Omron CX-Programmer project NewProject (CX-Programmer 9.61)

# PLC NewPLC1: CJ2M CPU11
I/O table (CPU CJ2M-CPU11): rack 0 slot 0 CJ1W-ID211; rack 0 slot 1 CJ1W-OD211

## Global symbols (name address type ; comment)
0.00 BOOL  ; PB Start
0.01 BOOL  ; PB Stop
0.02 BOOL  ; Emergency Stop
0.04 BOOL  ; Sensor C2PE
0.05 BOOL  ; PB1 C1
0.06 BOOL  ; PB2 C1
0.07 BOOL  ; Sensor STPX1
0.08 BOOL  ; Sensor STPX2
0.09 BOOL  ; Sensor STPX3
0.10 BOOL  ; Sensor PECA
0.11 BOOL  ; Sensor PECB
0.12 BOOL  ; Sensor PECC
0.14 BOOL  ; Sensor PEST
0.15 BOOL  ; Reset
1.00 BOOL  ; Conveyor C1
1.01 BOOL  ; Conveyor C2
1.02 BOOL  ; Light PBC1
1.03 BOOL  ; LIght PBC2
1.04 BOOL  ; Buzzer
1.06 BOOL  ; Conveyor ST2
1.07 BOOL  ; Coveyor CA
1.08 BOOL  ; Coveyor CB
1.09 BOOL  ; Conveyor CC
1.10 BOOL  ; Indikator Lampu CA
1.11 BOOL  ; Indikator Lampu CB
1.13 BOOL  ; Indikator Lampu CC
2.00 BOOL  ; System ON
2.01 BOOL  ; Memory 2
2.02 BOOL  ; Memory 3
2.03 BOOL  ; Masuk ke CA
2.04 BOOL  ; Masuk ke CB
2.05 BOOL  ; Masuk ke CC
D1 CHANNEL  ; Barcode Scanner
D100 CHANNEL  ; Data Barcode
D101 CHANNEL  ; Posisi Mobil
D102 CHANNEL  ; Conveyor ST2
T0000 BOOL  ; TB PBC2 UP
T0001 BOOL  ; TB PBC1 UP
T0002 BOOL  ; TB PBC2 DOWN
T0003 BOOL  ; TB PBC1 DOWN
T0004 BOOL  ; T BUZZ PB1/2 C1
T0005 BOOL  ; T BUZZ C15s
BarcodeProcess BarcodeScanner
Menentukan_Posisi_STPX SensorSTPX
Pengiriman PengirimanKeCACBCC

## Program SesiC (cyclic task 0)

### Section Main_Program

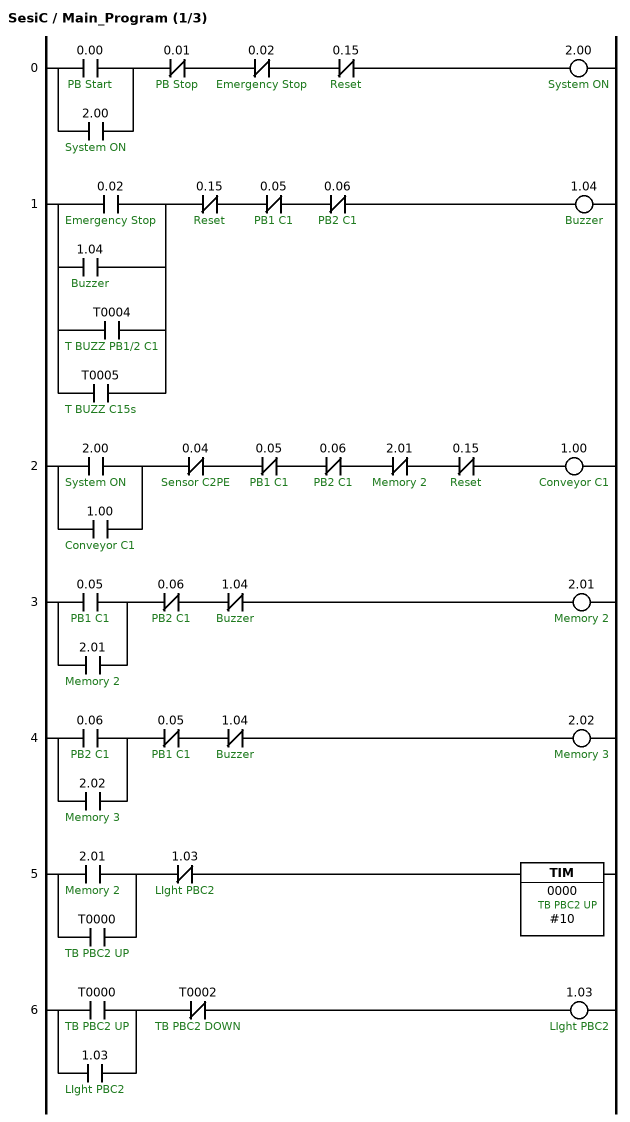
; rung 0
LD 0.00  ; PB Start
OR 2.00  ; System ON
ANDNOT 0.01  ; PB Stop
ANDNOT 0.02  ; Emergency Stop
ANDNOT 0.15  ; Reset
OUT 2.00  ; System ON
; rung 1
LD 0.02  ; Emergency Stop
OR 1.04  ; Buzzer
OR T0004  ; T BUZZ PB1/2 C1
OR T0005  ; T BUZZ C15s
ANDNOT 0.15  ; Reset
ANDNOT 0.05  ; PB1 C1
ANDNOT 0.06  ; PB2 C1
OUT 1.04  ; Buzzer
; rung 2
LD 2.00  ; System ON
OR 1.00  ; Conveyor C1
ANDNOT 0.04  ; Sensor C2PE
ANDNOT 0.05  ; PB1 C1
ANDNOT 0.06  ; PB2 C1
ANDNOT 2.01  ; Memory 2
ANDNOT 0.15  ; Reset
OUT 1.00  ; Conveyor C1
; rung 3
LD 0.05  ; PB1 C1
OR 2.01  ; Memory 2
ANDNOT 0.06  ; PB2 C1
ANDNOT 1.04  ; Buzzer
OUT 2.01  ; Memory 2
; rung 4
LD 0.06  ; PB2 C1
OR 2.02  ; Memory 3
ANDNOT 0.05  ; PB1 C1
ANDNOT 1.04  ; Buzzer
OUT 2.02  ; Memory 3
; rung 5
LD 2.01  ; Memory 2
OR T0000  ; TB PBC2 UP
ANDNOT 1.03  ; LIght PBC2
TIM 0000 #10  ; TB PBC2 UP
; rung 6
LD T0000  ; TB PBC2 UP
OR 1.03  ; LIght PBC2
ANDNOT T0002  ; TB PBC2 DOWN
OUT 1.03  ; LIght PBC2

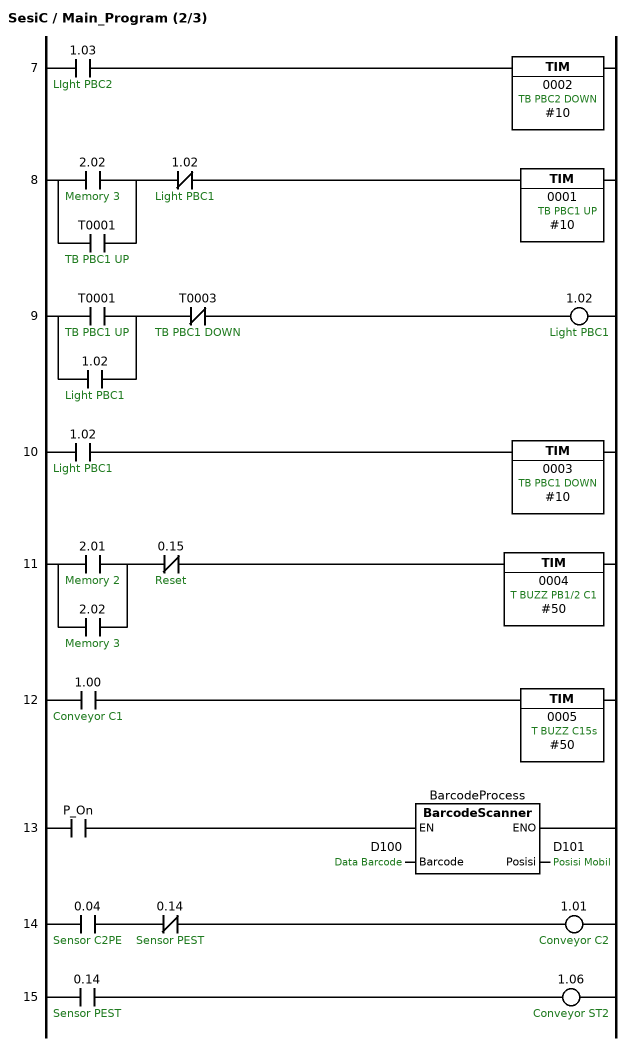
; rung 7
LD 1.03  ; LIght PBC2
TIM 0002 #10  ; TB PBC2 DOWN
; rung 8
LD 2.02  ; Memory 3
OR T0001  ; TB PBC1 UP
ANDNOT 1.02  ; Light PBC1
TIM 0001 #10  ; TB PBC1 UP
; rung 9
LD T0001  ; TB PBC1 UP
OR 1.02  ; Light PBC1
ANDNOT T0003  ; TB PBC1 DOWN
OUT 1.02  ; Light PBC1
; rung 10
LD 1.02  ; Light PBC1
TIM 0003 #10  ; TB PBC1 DOWN
; rung 11
LD 2.01  ; Memory 2
OR 2.02  ; Memory 3
ANDNOT 0.15  ; Reset
TIM 0004 #50  ; T BUZZ PB1/2 C1
; rung 12
LD 1.00  ; Conveyor C1
TIM 0005 #50  ; T BUZZ C15s
; rung 13
LD P_On
CALL BarcodeProcess : BarcodeScanner (Barcode := D100, Posisi => D101)  ; Data Barcode, Posisi Mobil
; rung 14
LD 0.04  ; Sensor C2PE
ANDNOT 0.14  ; Sensor PEST
OUT 1.01  ; Conveyor C2
; rung 15
LD 0.14  ; Sensor PEST
OUT 1.06  ; Conveyor ST2

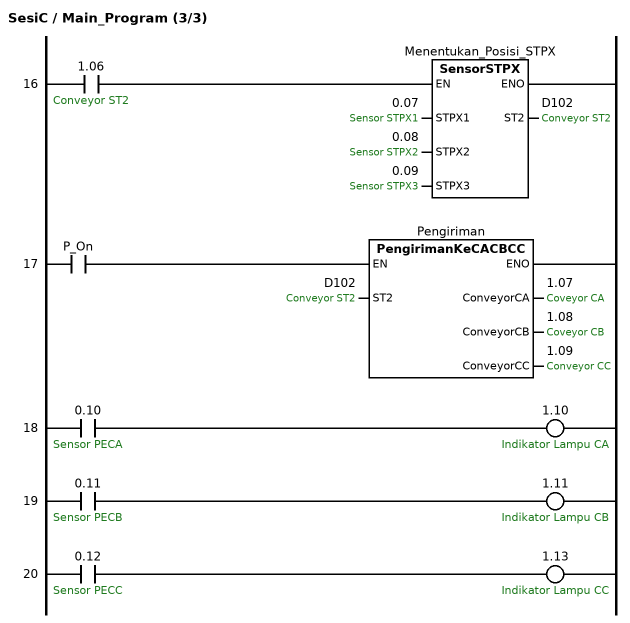
; rung 16
LD 1.06  ; Conveyor ST2
CALL Menentukan_Posisi_STPX : SensorSTPX (STPX1 := 0.07, STPX2 := 0.08, STPX3 := 0.09, ST2 => D102)  ; Sensor STPX1, Sensor STPX2, Sensor STPX3, Conveyor ST2
; rung 17
LD P_On
CALL Pengiriman : PengirimanKeCACBCC (ST2 := D102, ConveyorCA => 1.07, ConveyorCB => 1.08, ConveyorCC => 1.09)  ; Conveyor ST2, Coveyor CA, Coveyor CB, Conveyor CC
; rung 18
LD 0.10  ; Sensor PECA
OUT 1.10  ; Indikator Lampu CA
; rung 19
LD 0.11  ; Sensor PECB
OUT 1.11  ; Indikator Lampu CB
; rung 20
LD 0.12  ; Sensor PECC
OUT 1.13  ; Indikator Lampu CC

### Section END
; rung 0
END(001)

## Function block BarcodeScanner
VAR_INPUT
  Barcode : INT;
END_VAR
VAR_OUTPUT
  Posisi : INT;
END_VAR
IF Barcode = 1234 THEN Posisi:= 1;
ELSIF Barcode = 4321 THEN Posisi:= 2;
ELSIF Barcode = 2143 THEN Posisi:= 3;
END_IF;

## Function block PengirimanKeCACBCC
VAR_INPUT
  ST2 : INT;
END_VAR
VAR_OUTPUT
  ConveyorCA : BOOL;
  ConveyorCB : BOOL;
  ConveyorCC : BOOL;
END_VAR
IF ST2 = 1 THEN ConveyorCA:= TRUE;
ELSIF ST2 = 2 THEN ConveyorCB:= TRUE;
ELSIF ST2 = 3 THEN ConveyorCC:= TRUE;
END_IF;		

## Function block SensorSTPX
VAR_INPUT
  STPX1 : BOOL;
  STPX2 : BOOL;
  STPX3 : BOOL;
END_VAR
VAR_OUTPUT
  ST2 : INT;
END_VAR
IF (STPX1=TRUE AND STPX2=TRUE AND STPX3=FALSE) THEN ST2:= 1;
ELSIF (STPX1=TRUE AND STPX2=FALSE AND STPX3=TRUE) THEN ST2:= 2;
ELSIF (STPX1=FALSE AND STPX2=TRUE AND STPX3=TRUE) THEN ST2:= 3;
END_IF;